FUNCTION_BLOCK FB_Motion2way_Rodlock
VAR_INPUT
	
	//advances
	iAdvanceAuto: BOOL; //auto request
	iAdvanceManual: BOOL; //manual request
	iAdvanceInterlock: BOOL; //must be TRUE to perform motion
	iAdvanceDepth: BOOL; //limit sensor for advanced
	iAdvancePrompt: BOOL; //TRUE if the motion is the next step in the sequence


	iAdvanceTimeout:TIME := T#5S; //default timeout value
	
	//returns
	iReturnManual: BOOL; //manual request
	iReturnAuto: BOOL; //auto request
	iReturnInterlock: BOOL; //must be TRUE to perform motion
	iReturnTimeout:TIME := T#5S; //default timeout value
	iReturnDepth: BOOL; //limit sensor for advanced
	iReturnPrompt: BOOL; //TRUE if the motion is the next step in the sequence
	
	iLatchCoilOn: BOOL; //TRUE to latch the coil on after a motion
	
	iMode: typeStationMode; //what mode is station in?
	
	iRodlockTime:TIME:= T#250MS; //delay after rod lock release to perform motion

END_VAR
VAR_OUTPUT

	//advance coil
	qAdvanceCoil: BOOL;
	qAdvancedDepth: BOOL;
	qAdvanceTime: TIME;
	qAdvancePrompt: BOOL;
	qAdvanceInterlock: BOOL;
	
	//return coil
	qReturnCoil: BOOL;
	qReturnDepth: BOOL;
	qReturnTime: TIME;
	qReturnPrompt: BOOL;
	qReturnInterlock: BOOL;

	
	qFaultAdvanceTimeout: BOOL;		//TRUE if the advance switch was not reached
	qFaultReturnTimeout: BOOL;		//TRUE if the return switch was not reached
	qFaultLostAdvance: BOOL;		//TRUE if the advance switch was lost after advancing
	qFaultLostReturn: BOOL;			//TRUE if the return switch was lost after advancing
	qSwitchFault: BOOL;				//TRUE if Both the advance and return switch were TRUE
	
	qRodLock:BOOL;					//connect to raillock or rod lock output

END_VAR
VAR
	
	//advance variables
	tAdvanceReq: BOOL;
	timAdvanceTimer: TON;
	tAdvanceTimeoutFault: BOOL;
	tAdvanceWithInterlock: BOOL;
	
	//return variables
	tReturnReq: BOOL;
	timReturnTimer: TON;
	tReturnTimeoutFault: BOOL;
	tReturnWithInterlock: BOOL;
	
	
	timSwitchFault: TON;
	
	
	timRodLockRelease: TON;
	// Energise rodlock or raillock
	tEnableRodlock: BOOL;
END_VAR
VAR // added by the converter: edge detectors and wires of the graphical bodies
    _ft1, _ft2, _ft3, _ft4, _ft5, _ft6, _ft7 : F_TRIG;
    _w1, _w2 : BOOL;
END_VAR

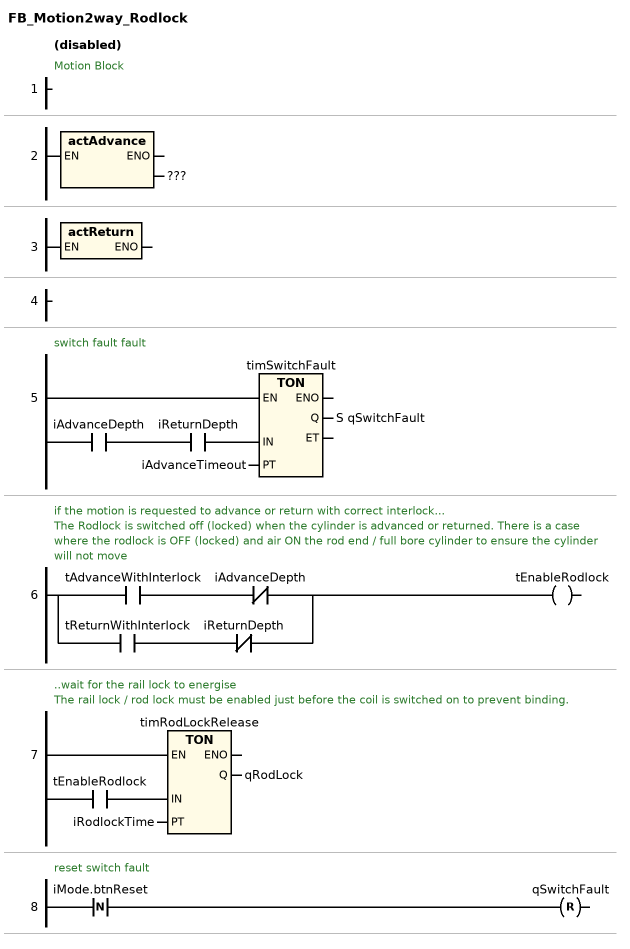
// NETWORK 1 (disabled)
// Motion Block

// NETWORK 2
actAdvance();

// NETWORK 3
actReturn();

// NETWORK 4

// NETWORK 5
// switch fault fault
timSwitchFault(IN := iAdvanceDepth AND iReturnDepth, PT := iAdvanceTimeout); // TON
qSwitchFault S= timSwitchFault.Q;

// NETWORK 6
// if the motion is requested to advance or return with correct interlock...
// The Rodlock is switched off (locked) when the cylinder is advanced or returned. There is a case where the rodlock is OFF (locked) and air ON the rod end / full bore cylinder to ensure the cylinder will not move
tEnableRodlock := tAdvanceWithInterlock AND NOT iAdvanceDepth OR tReturnWithInterlock AND NOT iReturnDepth;

// NETWORK 7
// ..wait for the rail lock to energise
// The rail lock / rod lock must be enabled just before the coil is switched on to prevent binding.
timRodLockRelease(IN := tEnableRodlock, PT := iRodlockTime, Q => qRodLock); // TON

// NETWORK 8
// reset switch fault
_ft1(CLK := iMode.btnReset);
qSwitchFault R= _ft1.Q;

ACTION actAdvance:
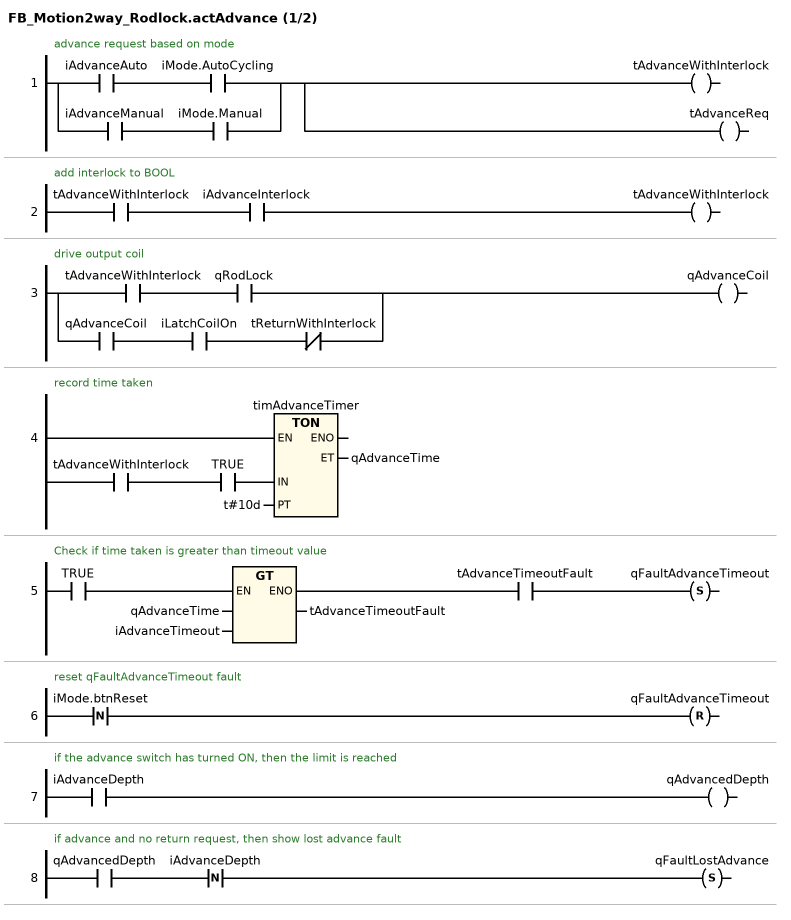
// NETWORK 1
// advance request based on mode
_w1 := iAdvanceAuto AND iMode.AutoCycling OR iAdvanceManual AND iMode.Manual;
tAdvanceWithInterlock := _w1;
tAdvanceReq := _w1;

// NETWORK 2
// add interlock to BOOL
tAdvanceWithInterlock := tAdvanceWithInterlock AND iAdvanceInterlock;

// NETWORK 3
// drive output coil
qAdvanceCoil := tAdvanceWithInterlock AND qRodLock OR qAdvanceCoil AND iLatchCoilOn AND NOT tReturnWithInterlock;

// NETWORK 4
// record time taken
timAdvanceTimer(IN := tAdvanceWithInterlock AND TRUE, PT := t#10d, ET => qAdvanceTime); // TON

// NETWORK 5
// Check if time taken is greater than timeout value
tAdvanceTimeoutFault := qAdvanceTime > iAdvanceTimeout;
qFaultAdvanceTimeout S= TRUE AND tAdvanceTimeoutFault;

// NETWORK 6
// reset qFaultAdvanceTimeout fault
_ft2(CLK := iMode.btnReset);
qFaultAdvanceTimeout R= _ft2.Q;

// NETWORK 7
// if the advance switch has turned ON, then the limit is reached
qAdvancedDepth := iAdvanceDepth;

// NETWORK 8
// if advance and no return request, then show lost advance fault
_ft3(CLK := iAdvanceDepth);
qFaultLostAdvance S= qAdvancedDepth AND _ft3.Q;

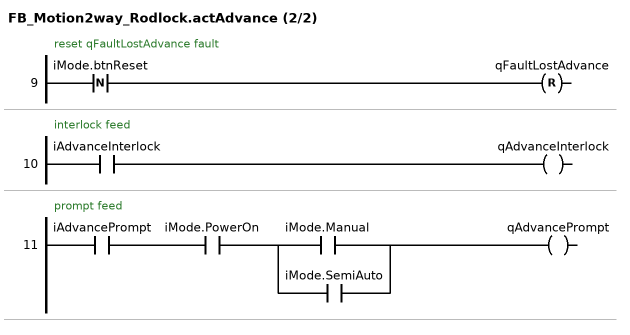
// NETWORK 9
// reset qFaultLostAdvance fault
_ft4(CLK := iMode.btnReset);
qFaultLostAdvance R= _ft4.Q;

// NETWORK 10
// interlock feed
qAdvanceInterlock := iAdvanceInterlock;

// NETWORK 11
// prompt feed
qAdvancePrompt := iAdvancePrompt AND iMode.PowerOn AND (iMode.Manual OR iMode.SemiAuto);
END_ACTION

ACTION actReturn:
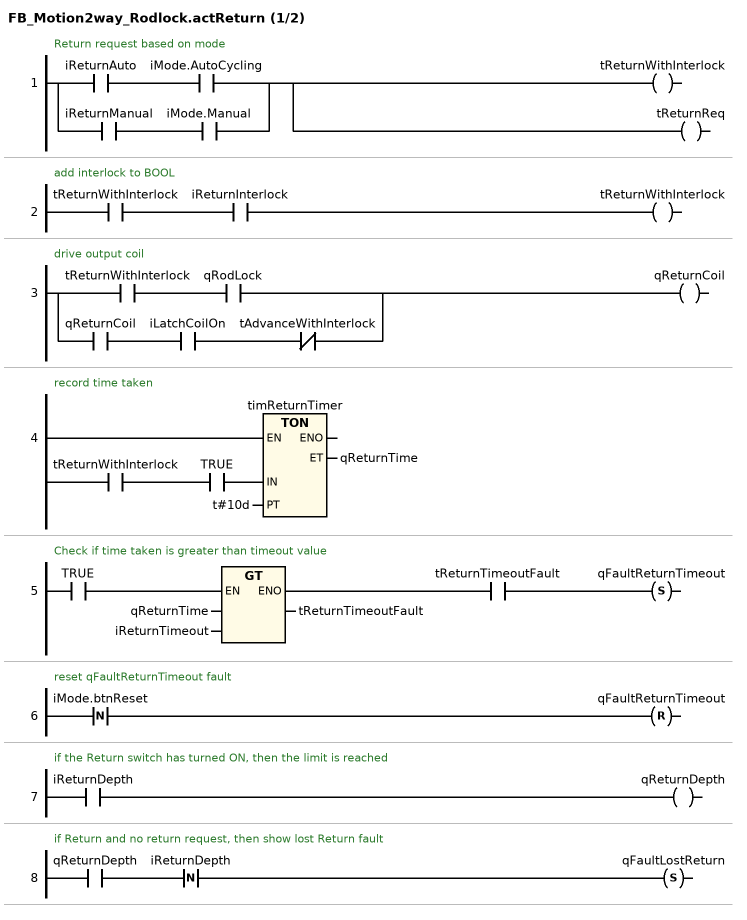
// NETWORK 1
// Return request based on mode
_w2 := iReturnAuto AND iMode.AutoCycling OR iReturnManual AND iMode.Manual;
tReturnWithInterlock := _w2;
tReturnReq := _w2;

// NETWORK 2
// add interlock to BOOL
tReturnWithInterlock := tReturnWithInterlock AND iReturnInterlock;

// NETWORK 3
// drive output coil
qReturnCoil := tReturnWithInterlock AND qRodLock OR qReturnCoil AND iLatchCoilOn AND NOT tAdvanceWithInterlock;

// NETWORK 4
// record time taken
timReturnTimer(IN := tReturnWithInterlock AND TRUE, PT := t#10d, ET => qReturnTime); // TON

// NETWORK 5
// Check if time taken is greater than timeout value
tReturnTimeoutFault := qReturnTime > iReturnTimeout;
qFaultReturnTimeout S= TRUE AND tReturnTimeoutFault;

// NETWORK 6
// reset qFaultReturnTimeout fault
_ft5(CLK := iMode.btnReset);
qFaultReturnTimeout R= _ft5.Q;

// NETWORK 7
// if the Return switch has turned ON, then the limit is reached
qReturnDepth := iReturnDepth;

// NETWORK 8
// if Return and no return request, then show lost Return fault
_ft6(CLK := iReturnDepth);
qFaultLostReturn S= qReturnDepth AND _ft6.Q;

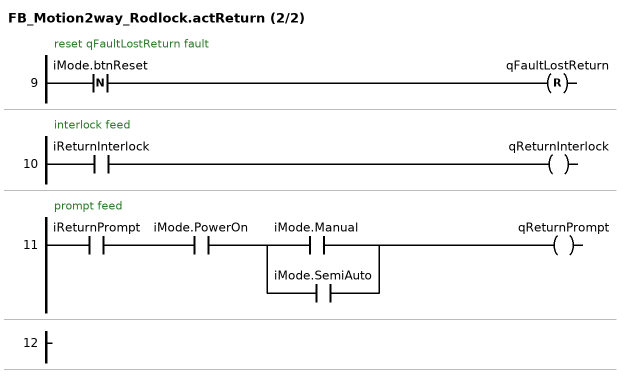
// NETWORK 9
// reset qFaultLostReturn fault
_ft7(CLK := iMode.btnReset);
qFaultLostReturn R= _ft7.Q;

// NETWORK 10
// interlock feed
qReturnInterlock := iReturnInterlock;

// NETWORK 11
// prompt feed
qReturnPrompt := iReturnPrompt AND iMode.PowerOn AND (iMode.Manual OR iMode.SemiAuto);

// NETWORK 12
END_ACTION

END_FUNCTION_BLOCK

(* stored: Version 1.1.0.1, ProductVersion 3.1.4024.12
   POU FB_Motion2way_Rodlock: Id {91059541-fa2d-4f29-90a8-bd9879d25195}, SpecialFunc None
   Action actAdvance: Id {46f4bd58-5ce0-491e-8278-1ea76200a1c3}
   Action actReturn: Id {9ac35b85-3aef-4518-8c6f-7f27c1694504} *)
